// TwinCAT 3 PLC project PLC1
// ProgramVersion: 3.1.4024.0
// libraries:
//   Tc2_Standard, * (Beckhoff Automation GmbH)
//   Tc2_System, * (Beckhoff Automation GmbH)
//   Tc3_Module, * (Beckhoff Automation GmbH)
//   VisuSymbols,3.5.10.0,System
// project tree:
//   DUTs/ E_States.TcDUT, ST_Sensor.TcDUT
//   / GlobalTextList.TcGTLO, PlcTask.TcTTO, Visualization Manager.TcVMO (not stored)
//   GVLs/ GVL.TcGVL
//   POUs/ ArrayStorage.TcPOU, Case_Chase.TcPOU, Class Diagram.TcCD (not stored), FB_Blink182.TcPOU, F_Scaling.TcPOU, F_ScalingByRef.TcPOU, MAIN.TcPOU, StructureTesting.TcPOU
//   VISUs/ Visualization.TcVIS
// real-time tasks:
//   TASK PlcTask: cycle T#10ms, priority 20, ADS port 350
// motion (NC):
//   TASK NC-Task 1 SAF: cycle T#2ms, priority 4, ADS port 501
//   TASK NC-Task 1 SVB: cycle T#10ms, priority 8, ADS port 511
//   AXIS Axis 1 (id 1)
//     General: UnitName=Degree
//     Dynamic: Acceleration=14535, Deceleration=14535, Jerk=43605
//     Velo: RefSearch=96.9, RefSync=96.9, SlowManual=484.5, FastManual=2907, Fast=9690, Maximum=9690
//     OtherSettings: AllowMotionCmdToSlave=true
//     encoder EncType=19
//       EncPara: ScaleFactorNumerator=360, ScaleFactorDenominator=1048576, EncMode=3, MaxCount=#xffffffff
//     drive DrvType=16
//       DrvPara: MaxCount=#xffffffff, DriveControlDWord=#x00020100
//         Analog: VeloReferenz=10659, VeloScale=32, TorqueSetpointScale=10, ScaleFactorActTorque=0.1
//         TimeComp: TaskDelayCycles=1
//     controller CtrType=1
//       CtrPara: PriorControlFactor=1
//         PosDiffControl: Range=50
//         Observer: BandWidth=20
// I/O:
//   DEVICE Device 1 (EtherCAT), AmsNetId 5.135.114.183.2.1
//     Term 1 (EK1200) [EK1200-5000 EtherCAT Power supply (2A E-Bus)]
//       Term 2 (EL1859) [EL1859 8Ch. Dig. Input 24V, 3ms, 8Ch. Dig. Output 24V, 0.5A]
//       Term 3 (EL1859) [EL1859 8Ch. Dig. Input 24V, 3ms, 8Ch. Dig. Output 24V, 0.5A]
//       Term 4 (EL3255) [EL3255 5Ch. potentiometer measurement with sensor supply]
//       Term 5 (EL3214-0090) [EL3214-0090 4Ch. Ana. Input PT100 (RTD), TwinSAFE SC]
//       Term 6 (EL5151) [EL5151 1Ch. Inc. Encoder]
//       Term 7 (EL1918) [EL1918, 8Ch. Safety Input 24V, TwinSAFE]
//         modules: Module 1 (FSOE), Module 2 (FSLOGIC)
//       Term 8 (EL2912) [EL2912, 2Ch. Safety Output 24V, 2A, TwinSAFE]
//         modules: Module 1 (FSOE), Module 2 (FSOUT), Module 3 (DEVICEIO), Module 4 (FSLOGIC)
//       Term 9 (EL9110) [EL9110 Power Supplier with LED (24V, Diagnostics)]
//       Term 10 (EL7201-9014) [EL7201-9014 1Ch. MDP742 Servo motor output stage with OCT (50V, 2.8A RMS) and STO input]
//       Term 11 (EK1122) [EK1122 2 port EtherCAT junction]
//       Term 12 (EL9011) [EL9011 End Terminal]
//   DEVICE Device 3 (EtherCAT Automation Protocol), AmsNetId 5.135.114.183.4.1
//     Box 13 (Publisher)
//     Box 14 (Subscriber)
//     Box 15 (Subscriber)
// variable links:
//   NC-Task 1 SAF/Axes/Axis 1 <-> Device 1 (EtherCAT)/Term 1 (EK1200)/Term 10 (EL7201-9014)
//     Drive/Inputs/In/nDataIn1 <-> DRV Following error actual value/Following error actual value
//     Drive/Inputs/In/nDataIn3[0] <-> DRV Torque actual value/Torque actual value
//     Drive/Inputs/In/nDcOutputTime <-> InfoData/DcOutputShift
//     Drive/Inputs/In/nState1 <-> DRV Statusword/Statusword
//     Drive/Inputs/In/nState2 <-> DRV Statusword/Statusword @bit 8
//     Drive/Inputs/In/nState4 @bit 1 <-> WcState/InputToggle
//     Drive/Inputs/In/nState4 <-> WcState/WcState
//     Drive/Outputs/Out/nCtrl1 <-> DRV Controlword/Controlword
//     Drive/Outputs/Out/nCtrl2 <-> DRV Controlword/Controlword @bit 8
//     Drive/Outputs/Out/nDataOut1 <-> DRV Target position/Target position
//     Enc/Inputs/In/nDataIn1 <-> FB Position/Position
//     Enc/Inputs/In/nDcInputTime <-> InfoData/DcInputShift
//     Enc/Inputs/In/nState4 @bit 1 <-> WcState/InputToggle
//     Enc/Inputs/In/nState4 <-> WcState/WcState
//   PLC1/PLC1 Instance <-> Device 1 (EtherCAT)/Term 1 (EK1200)/Term 2 (EL1859)
//     PlcTask Inputs/GVL.aSwitches[{1..8}] <-> Channel {1..8}/Input  (8 links)
//     PlcTask Outputs/GVL.aLights[{1..8}] <-> Channel {9..16}/Output  (8 links)
//   PLC1/PLC1 Instance <-> Device 1 (EtherCAT)/Term 1 (EK1200)/Term 3 (EL1859)
//     PlcTask Inputs/GVL.bReset <-> Channel 1/Input
//   PLC1/PLC1 Instance <-> Device 1 (EtherCAT)/Term 1 (EK1200)/Term 4 (EL3255)
//     PlcTask Inputs/GVL.iPot1 <-> AI Standard Channel 1/Value
//     PlcTask Inputs/StructureTesting.aSensors[1].rawTemp <-> AI Standard Channel 1/Value
//   PLC1/PLC1 Instance <-> Device 1 (EtherCAT)/Term 1 (EK1200)/Term 5 (EL3214-0090)
//     PlcTask Inputs/GVL.iPot2 <-> RTD Inputs Channel 1/Value
//     PlcTask Inputs/StructureTesting.aSensors[2].rawTemp <-> RTD Inputs Channel 1/Value
//   PLC1/PLC1 Instance <-> Device 3 (EtherCAT Automation Protocol)/Box 13 (Publisher)
//     PlcTask Outputs/MAIN.ipot1OutputJeanPaul <-> Pub-Var 1/Outputs/VarData

CONFIGURATION PLC1
    RESOURCE PLC ON TwinCAT3
        TASK PlcTask(INTERVAL := T#10ms, PRIORITY := 20);
        PROGRAM MAIN WITH PlcTask : MAIN;
    END_RESOURCE
END_CONFIGURATION

// ---- DUTs/E_States.TcDUT
{attribute 'qualified_only'}
{attribute 'strict'}
TYPE E_States :
(
	oneSecondPress := 100,
	threeCountPress := 200,
	twoButtonPress := 300,
	blinkingLight := 400,
	oneSecondRelease := 410
);
END_TYPE

// ---- DUTs/ST_Sensor.TcDUT
TYPE ST_Sensor :
STRUCT
	rawTemp AT %I* : INT;
	scaledTemp : REAL;
END_STRUCT
END_TYPE

// ---- GVLs/GVL.TcGVL
{attribute 'qualified_only'}
VAR_GLOBAL
	aSwitches 	AT %I* : ARRAY [1..8]OF BOOL;
	aLights 	AT %Q* : ARRAY [1..8]OF BOOL;
	iPot1 		AT %I* : INT;
	iPot2		AT %I* : INT;
	bReset		AT %I* : BOOL;
END_VAR

// ---- POUs/MAIN.TcPOU
PROGRAM MAIN
VAR
	ipot1OutputJeanPaul AT %Q* :INT;
END_VAR

 ArrayStorage();
 Case_Chase();
 StructureTesting();
 
 ipot1OutputJeanPaul := gvl.iPot1;

END_PROGRAM

// ---- POUs/ArrayStorage.TcPOU
PROGRAM ArrayStorage
VAR
	aPotValues : ARRAY [lowBound..highBound] OF INT ;
	i: INT :=1;
	ftrig1: F_TRIG;
	rtrig1: R_TRIG;
END_VAR

VAR CONSTANT
	lowBound : 	INT := 1;
	highBound : INT := 5;
END_VAR

IF GVL.aSwitches[1] AND i>=lowBound AND i<=highBound THEN 
	aPotValues[i] := GVL.iPot1;
END_IF

ftrig1(CLK:= GVL.aSwitches[1]);


IF ftrig1.Q AND i>=lowBound AND i<highBound THEN
	i := i+1;
END_IF

IF gvl.bReset THEN
	FOR i:= lowBound TO highBound DO
		aPotValues[i] := 0;
	END_FOR
	i := lowBound;
	END_IF
	
rtrig1(CLK:= GVL.aSwitches[2]);
	
IF rtrig1.Q THEN
	i := i-1;
	IF i>= lowBound AND i<= highBound THEN
		aPotValues[i] := 0;
	END_IF
	IF i < lowBound THEN
		i := lowBound;
	END_IF
END_IF

END_PROGRAM

// ---- POUs/Case_Chase.TcPOU
PROGRAM Case_Chase
VAR
	iState : E_STATES;
	ton1: TON;
	ton2: TON;
	ton3: TON;
	ton4: TON;
	fbCTU23: CTU;
	fb_blink182: FB_Blink182;
	f_trig400: F_TRIG;
END_VAR

CASE iState OF
E_States.oneSecondPress:
		ton1.IN:= GVL.aSwitches[5]; 
		ton1.PT:=T#1S;
		GVL.aLights[5] := 1;
		IF ton1.Q = 1 THEN
			ton1.IN:=0;
			iState := E_States.threeCountPress; 
			GVL.aLights[5] := 0;
		END_IF
E_States.threeCountPress:
		GVL.aLights[6] := 1;
		fbCTU23.CU := GVL.aSwitches[6];
		fbCTU23(PV :=3);
		fbCTU23(RESET := FALSE);
		//ton2.IN:= GVL.aSwitches[6]; 
		//ton2.PT:=T#1S;
		IF fbCTU23.Q = 1 THEN
			//ton2.IN:=0;
			iState := E_States.twoButtonPress; 
			GVL.aLights[6] := 0;
			fbCTU23(RESET := TRUE);
		END_IF 
E_States.twoButtonPress:
		//ton3.IN:= GVL.aSwitches[7]; 
		//ton3.PT:=T#1S;
		GVL.aLights[7] := 1;
		IF GVL.aSwitches[5] AND GVL.aSwitches[6] THEN
			//ton3.IN:=0;
			iState := E_States.blinkingLight; 
			GVL.aLights[7]:= 0;
		END_IF
E_States.blinkingLight:
		fb_blink182(in:= NOT GVL.aSwitches[8], blink182PerSecond:= 2, Q=> GVL.aLights[8] );
		IF GVL.aSwitches[8] THEN
			iState := E_States.oneSecondRelease;
		END_IF
		
E_States.oneSecondRelease: 
		GVL.aLights[8] := TRUE;
		 IF NOT GVL.aSwitches[8] THEN
			ton4(IN := TRUE);
			ton4(PT:=T#1S);
		END_IF
			
		IF 	ton4.Q = TRUE THEN
			ton4(IN := FALSE);
			GVL.aLights[8] := FALSE;
			iState := E_States.oneSecondPress;
			
		END_IF
END_CASE

ton1();
ton2();
ton3();
ton4();

END_PROGRAM

// ---- POUs/FB_Blink182.TcPOU
FUNCTION_BLOCK FB_Blink182
VAR_INPUT
	in : BOOL;
	blink182PerSecond : INT;
END_VAR

VAR_OUTPUT
	Q : BOOL;
END_VAR

VAR
	pulse1: TON;
END_VAR

pulse1(IN:= in , PT:= T#1S/(blink182PerSecond*2) , Q=>  , ET=> );

IF pulse1.Q THEN
	Q := NOT Q;
	pulse1(IN:= FALSE);
END_IF

END_FUNCTION_BLOCK

// ---- POUs/StructureTesting.TcPOU
PROGRAM StructureTesting
VAR
	aSensors : ARRAY[1..2] OF ST_Sensor;
END_VAR

//aSensors[1].scaledTemp := (aSensors[1].rawTemp)/327.67;
//aSensors[2].scaledTemp := (aSensors[2].rawTemp)/

aSensors[1].scaledTemp := F_Scaling(rawInput:= aSensors[1].rawTemp );

END_PROGRAM

// ---- POUs/F_Scaling.TcPOU
FUNCTION F_Scaling : REAL
VAR_INPUT
	rawInput : INT;
END_VAR
VAR
END_VAR

F_Scaling := rawInput/327.67;

END_FUNCTION

// ---- POUs/F_ScalingByRef.TcPOU
FUNCTION F_ScalingByRef : BOOL
VAR_INPUT
	entireSensor : REFERENCE TO ST_Sensor;
END_VAR
VAR
END_VAR

IF entireSensor.rawTemp >=0 THEN
	entireSensor.scaledTemp := (entireSensor.rawTemp/327.67);
	F_ScalingByRef := TRUE;
	RETURN;
ELSE
	F_ScalingByRef:=FALSE;
	
END_IF

END_FUNCTION

// ---- VISUs/Visualization.TcVIS
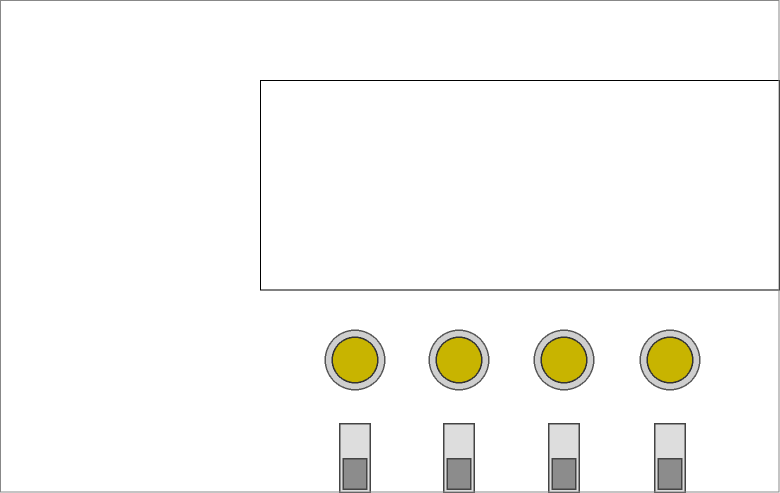
VISUALIZATION Visualization  // 780x493
    Rectangle (260,80 520x210)
    DipSwitch (320,423 70x70), variable: GVL.aSwitches[5], behaviour: TOGGLE, style: Switch-DipSwitch-Gray
    Lamp1 (320,325 70x70), variable: GVL.aLights[5], style: Lamp-Lamp1-Yellow
    DipSwitch (424,423 70x70), variable: GVL.aSwitches[6], behaviour: TOGGLE, style: Switch-DipSwitch-Gray
    Lamp1 (424,325 70x70), variable: GVL.aLights[6], style: Lamp-Lamp1-Yellow
    DipSwitch (529,423 70x70), variable: GVL.aSwitches[7], behaviour: TOGGLE, style: Switch-DipSwitch-Gray
    Lamp1 (529,325 70x70), variable: GVL.aLights[7], style: Lamp-Lamp1-Yellow
    DipSwitch (635,423 70x70), variable: GVL.aSwitches[8], behaviour: TOGGLE, style: Switch-DipSwitch-Gray
    Lamp1 (635,325 70x70), variable: GVL.aLights[8], style: Lamp-Lamp1-Yellow
END_VISUALIZATION
